{attribute 'qualified_only'}
{attribute 'strict'}
TYPE E_SpeedModeLocalController_EMS :
(
	eSlow			:= 0,
	eBalanced 		:= 1,
	eFast			:= 2
);
END_TYPE

(* stored: Version 1.1.0.1, ProductVersion 3.1.4024.9
   DUT E_SpeedModeLocalController_EMS: Id {076ec630-c16e-4748-b9f2-0a8e1e705e48} *)
